TYPE TcoRotaryTransfer_Status EXTENDS TcoCore.TcoStruct:
STRUCT


		ActionDescription:STRING;
		
END_STRUCT
END_TYPE

(* stored: Version 1.1.0.1
   DUT TcoRotaryTransfer_Status: Id {6066b0c7-22fb-4319-964d-f99e5997d80b} *)
